(* PLC project RobotLibrary, Beckhoff Automation GmbH TwinCAT PLC Control 3.5.13.21 *)
(* stored: creationDateTime 2024-06-05T21:41:09.5070225, modificationDateTime 2024-06-05T21:41:09.5090704 *)

{attribute 'pack_mode' := '1'} 
// ------------------------------------------------------------------------- 
//  SRCI Robot Library                                                
// ------------------------------------------------------------------------- 
//                                                                           
//  Object:      ExecutionModeAllowed                                       
//  Author:      Thorsten Brach                                                
//  Date:        2024-06-01
//
//  Description:                                              
//   
//                                                                           
//  Copyright: 
//    (C) 2024 Thorsten Brach. All rights reserved                                                                         
//                                                                           
//  Disclaimer:                                                                           
//    This project is provided without any guarantee and can be used for   
//    private and commercial purposes. Any commercial use is at the user’s 
//    own risk and responsibility.
//
// -------------------------------------------------------------------------
TYPE ExecutionModeAllowed :
STRUCT
  ///
  PRIMARY_SEQ         : BOOL;
  ///
  PRIMARY_SEQ_ABORT   : BOOL;
  ///
  SECONDARY_SEQ       : BOOL;
  ///
  SECONDARY_SEQ_ABORT : BOOL;
  ///
  PAR                 : BOOL := TRUE;
  ///
  PAR_TASK            : BOOL;
  ///
  PAR_TRIGGER         : BOOL;
  ///
  PAR_TRIGGER_TASK    : BOOL;
END_STRUCT
END_TYPE

{attribute 'pack_mode' := '1'} 
// ------------------------------------------------------------------------- 
//  SRCI Robot Library                                                
// ------------------------------------------------------------------------- 
//                                                                           
//  Object:      MessageHeaderCommand                                       
//  Author:      Thorsten Brach                                                
//  Date:        2024-06-01
//
//  Description:                                              
//   
//                                                                           
//  Copyright: 
//    (C) 2024 Thorsten Brach. All rights reserved                                                                         
//                                                                           
//  Disclaimer:                                                                           
//    This project is provided without any guarantee and can be used for   
//    private and commercial purposes. Any commercial use is at the user’s 
//    own risk and responsibility.
//
// -------------------------------------------------------------------------
TYPE MessageHeaderCommand :
STRUCT
  /// Byte 00-01 :  CMD type as per specification
  CmdType      : CmdType;
  /// Byte 02  : ExecutionMode (Bit 0..3)
  ExecMode     : BYTE;  
  /// Byte 03 : CMD priority (Bit 0..3)
  Prio         : BYTE;
  /// Byte 03 : Parameter Sequence (Bit 4..7 )
  ParSeq       : BYTE;
  /// Trigger related EmitterID
  EmitterID    : ARRAY[0..3] OF SINT;
  /// Trigger related ListenerID 
  ListenerID   : SINT;
  /// Reserved
  Reserved     : BYTE;
  //// Payload length defined by type per CMD definition. Processed by Appl. Layer Task.
  Payload      : ARRAY[0..RobotLibraryParameter.TELEGRAM_PAYLOAD_MAX] OF BYTE;  
END_STRUCT
END_TYPE

{attribute 'pack_mode' := '1'} 
// ------------------------------------------------------------------------- 
//  SRCI Robot Library                                                
// ------------------------------------------------------------------------- 
//                                                                           
//  Object:      MessageHeaderResponse                                       
//  Author:      Thorsten Brach                                                
//  Date:        2024-06-01
//
//  Description:                                              
//   
//                                                                           
//  Copyright: 
//    (C) 2024 Thorsten Brach. All rights reserved                                                                         
//                                                                           
//  Disclaimer:                                                                           
//    This project is provided without any guarantee and can be used for   
//    private and commercial purposes. Any commercial use is at the user’s 
//    own risk and responsibility.
//
// -------------------------------------------------------------------------
TYPE MessageHeaderResponse :
STRUCT
  /// Byte 03 : CMD priority (Bit 0..3)
  Prio                    : BYTE;
  /// Byte 03 : Parameter Sequence (Bit 4..7 )
  ParSeq                  : BYTE;
  /// Alarm Message Severity
  AlarmMessageSeverity    : Severity;
  /// Alarm Message Code
  AlarmMessageCode        : UINT;
  /// Number of Trigger based CMD invocations
  InvocationCounter       : USINT;
  /// Number of missed Triggers
  MissedInvocationCounter : USINT;
  /// FollowID of Trigger initiator
  OriginID                : WORD;
  /// RSP Payload defined by type per CMD definition. Generated by Appl. Layer Task
  Payload                 : ARRAY[0..RobotLibraryParameter.TELEGRAM_PAYLOAD_MAX] OF BYTE;  
END_STRUCT
END_TYPE

{attribute 'qualified_only'}
// ------------------------------------------------------------------------- 
//  SRCI Robot Library                                                
// ------------------------------------------------------------------------- 
//                                                                           
//  Object:      ArmConfigElbow                                       
//  Author:      Thorsten Brach                                                
//  Date:        2024-06-01
//
//  Description:                                              
//   
//                                                                           
//  Copyright: 
//    (C) 2024 Thorsten Brach. All rights reserved                                                                         
//                                                                           
//  Disclaimer:                                                                           
//    This project is provided without any guarantee and can be used for   
//    private and commercial purposes. Any commercial use is at the user’s 
//    own risk and responsibility.
//
// -------------------------------------------------------------------------
TYPE ArmConfigElbow :
(
 /// Use config in position	
 USE_CONFIG := 0,
 /// Do not change config with this movement. (default)
 SAME := 1,
 /// Configuration in position is not used but the Robot is free to change config
 FREE := 2,
 /// Set elbow configuration in position to Down
 DOWN := 3,
 /// Set elbow configuration in position to up
 UP   := 4
);
END_TYPE

{attribute 'qualified_only'}
// ------------------------------------------------------------------------- 
//  SRCI Robot Library                                                
// ------------------------------------------------------------------------- 
//                                                                           
//  Object:      ArmConfigShoulder                                       
//  Author:      Thorsten Brach                                                
//  Date:        2024-06-01
//
//  Description:                                              
//   
//                                                                           
//  Copyright: 
//    (C) 2024 Thorsten Brach. All rights reserved                                                                         
//                                                                           
//  Disclaimer:                                                                           
//    This project is provided without any guarantee and can be used for   
//    private and commercial purposes. Any commercial use is at the user’s 
//    own risk and responsibility.
//
// -------------------------------------------------------------------------
TYPE ArmConfigShoulder :
(
 /// Use config in position	
 USE_CONFIG := 0,
 /// Do not change config with this movement. (default)
 SAME := 1,
 /// Configuration in position is not used but the Robot is free to change config
 FREE := 2,
 /// Set shoulder configuration in position to Back
 BACK := 3,
 /// Set shoulder configuration in position to Front
 FRONT := 4
);
END_TYPE

{attribute 'qualified_only'}
// ------------------------------------------------------------------------- 
//  SRCI Robot Library                                                
// ------------------------------------------------------------------------- 
//                                                                           
//  Object:      ArmConfigWrist                                       
//  Author:      Thorsten Brach                                                
//  Date:        2024-06-01
//
//  Description:                                              
//   
//                                                                           
//  Copyright: 
//    (C) 2024 Thorsten Brach. All rights reserved                                                                         
//                                                                           
//  Disclaimer:                                                                           
//    This project is provided without any guarantee and can be used for   
//    private and commercial purposes. Any commercial use is at the user’s 
//    own risk and responsibility.
//
// -------------------------------------------------------------------------
TYPE ArmConfigWrist :
(
 /// Use config in position	
 USE_CONFIG := 0,
 /// Do not change config with this movement. (default)
 SAME := 1,
 /// Configuration in position is not used but the Robot is free to change config
 FREE := 2,
 /// Set wrist configuration in position to Flip
 FLIP := 3,
 /// Set wrist configuration in position to Non-Flip
 NON_FLIP := 4
);
END_TYPE

{attribute 'qualified_only'}
// ------------------------------------------------------------------------- 
//  SRCI Robot Library                                                
// ------------------------------------------------------------------------- 
//                                                                           
//  Object:      SequenceFlag                                       
//  Author:      Thorsten Brach                                                
//  Date:        2024-06-01
//
//  Description:                                              
//   
//                                                                           
//  Copyright: 
//    (C) 2024 Thorsten Brach. All rights reserved                                                                         
//                                                                           
//  Disclaimer:                                                                           
//    This project is provided without any guarantee and can be used for   
//    private and commercial purposes. Any commercial use is at the user’s 
//    own risk and responsibility.
//
// -------------------------------------------------------------------------
TYPE SequenceFlag :
(
  /// • Refers to ProcessingModes 2 to 5 and 9
  /// • Command is not handled by any sequence
  /// • For more information on ProcessingModes refer to chapter 5.6.4.5
	NO_SEQUENCE        := 0,
  /// • Command will be handled by primary sequence
  PRIMARY_SEQUENCE   := 1,
  /// • Command will be handled by secondary sequence
  SECONDARY_SEQUENCE := 2
)USINT;
END_TYPE

{attribute 'qualified_only'}
// ------------------------------------------------------------------------- 
//  SRCI Robot Library                                                
// ------------------------------------------------------------------------- 
//                                                                           
//  Object:      LogLevel                                       
//  Author:      Thorsten Brach                                                
//  Date:        2024-06-01
//
//  Description:                                              
//   
//                                                                           
//  Copyright: 
//    (C) 2024 Thorsten Brach. All rights reserved                                                                         
//                                                                           
//  Disclaimer:                                                                           
//    This project is provided without any guarantee and can be used for   
//    private and commercial purposes. Any commercial use is at the user’s 
//    own risk and responsibility.
//
// -------------------------------------------------------------------------
TYPE LogLevel  :
(
  /// No events will be logged
  DEACTIVATE  := 0,
  /// Debugging messages, Informative messages, Warning messages, Error messages, Fatal error messages 
  DEBUG       := 4,
  /// Informative messages, Warning messages, Error messages, Fatal error messages
  INFO        := 5, 
  /// Warning messages, Error messages, Fatal error messages
  WARNING     := 20,
  /// Error messages, Fatal error messages 
  ERROR       := 28, 
  /// Fatal error messages
  FATAL_ERROR := 29 
)USINT;
END_TYPE

{attribute 'qualified_only'}
// ------------------------------------------------------------------------- 
//  SRCI Robot Library                                                
// ------------------------------------------------------------------------- 
//                                                                           
//  Object:      MessageLevel                                       
//  Author:      Thorsten Brach                                                
//  Date:        2024-06-01
//
//  Description:                                              
//   
//                                                                           
//  Copyright: 
//    (C) 2024 Thorsten Brach. All rights reserved                                                                         
//                                                                           
//  Disclaimer:                                                                           
//    This project is provided without any guarantee and can be used for   
//    private and commercial purposes. Any commercial use is at the user’s 
//    own risk and responsibility.
//
// -------------------------------------------------------------------------
TYPE MessageLevel :
(
  /// Debugging messages, Informative messages, Warning messages, Error messages, Fatal error messages
	DEBUG := 4,
  /// Informative messages, Warning messages, Error messages, Fatal error messages 
  INFO := 5, 
  /// Warning messages, Error messages, Fatal error messages
  WARNING := 20,
  /// Error messages, Fatal error messages 
  ERROR := 28 
)USINT;
END_TYPE

{attribute 'qualified_only'}
// ------------------------------------------------------------------------- 
//  SRCI Robot Library                                                
// ------------------------------------------------------------------------- 
//                                                                           
//  Object:      PriorityLevel                                       
//  Author:      Thorsten Brach                                                
//  Date:        2024-06-01
//
//  Description:                                              
//   
//                                                                           
//  Copyright: 
//    (C) 2024 Thorsten Brach. All rights reserved                                                                         
//                                                                           
//  Disclaimer:                                                                           
//    This project is provided without any guarantee and can be used for   
//    private and commercial purposes. Any commercial use is at the user’s 
//    own risk and responsibility.
//
// -------------------------------------------------------------------------
TYPE PriorityLevel :
(
  /// priority level is very high 
	VERY_HIGH := 1,
  /// priority level is high 
  HIGH      := 2,
  /// priority level is normal 
	NORMAL    := 3,
  /// priority level is low 
	LOW       := 4  
)BYTE;
END_TYPE

{attribute 'qualified_only'}
{attribute 'strict'}
// ------------------------------------------------------------------------- 
//  SRCI Robot Library                                                
// ------------------------------------------------------------------------- 
//                                                                           
//  Object:      CircPlane                                       
//  Author:      Thorsten Brach                                                
//  Date:        2024-06-01
//
//  Description:                                              
//   
//                                                                           
//  Copyright: 
//    (C) 2024 Thorsten Brach. All rights reserved                                                                         
//                                                                           
//  Disclaimer:                                                                           
//    This project is provided without any guarantee and can be used for   
//    private and commercial purposes. Any commercial use is at the user’s 
//    own risk and responsibility.
//
// -------------------------------------------------------------------------
TYPE CircPlane :
(
  /// x-z-plane
	XZ_PLANE := 0,
  /// y-z-plane
  YZ_PLANE := 1,
  /// x-y-plane
  XY_PLANE := 2
)SINT;
END_TYPE

{attribute 'qualified_only'}
// ------------------------------------------------------------------------- 
//  SRCI Robot Library                                                
// ------------------------------------------------------------------------- 
//                                                                           
//  Object:      ControlHalfByte                                       
//  Author:      Thorsten Brach                                                
//  Date:        2024-06-01
//
//  Description:                                              
//   
//                                                                           
//  Copyright: 
//    (C) 2024 Thorsten Brach. All rights reserved                                                                         
//                                                                           
//  Disclaimer:                                                                           
//    This project is provided without any guarantee and can be used for   
//    private and commercial purposes. Any commercial use is at the user’s 
//    own risk and responsibility.
//
// -------------------------------------------------------------------------
TYPE ControlHalfByte :
(
  /// Default value, no control active
  NONE := 0,
  /// Initialization is requested by the client
  INITIALIZE := 1,
  /// Resume of operation is requested by the client
  RESUME := 2,
  /// Resetting of the RC is requested by the client. The RC must stop the motion, and clear all state.
  RESET := 3,
  /// Acknowledgement of a telegram state error
  ACK_ERROR := 4,
  /// Signaling that a client error occurred. The Server must respond by setting its RI state to NOT_INITIALIZED
  CLIENT_ERROR := 5
)BYTE;
END_TYPE

{attribute 'qualified_only'}
// ------------------------------------------------------------------------- 
//  SRCI Robot Library                                                
// ------------------------------------------------------------------------- 
//                                                                           
//  Object:      ErrorReaction                                       
//  Author:      Thorsten Brach                                                
//  Date:        2024-06-01
//
//  Description:                                              
//   
//                                                                           
//  Copyright: 
//    (C) 2024 Thorsten Brach. All rights reserved                                                                         
//                                                                           
//  Disclaimer:                                                                           
//    This project is provided without any guarantee and can be used for   
//    private and commercial purposes. Any commercial use is at the user’s 
//    own risk and responsibility.
//
// -------------------------------------------------------------------------
TYPE ErrorReaction :
(
  /// Abort and move Abort active move command and delete commands buffered in sequence Move robot by specified ErrorVector
  ABORT_AND_MOVE := 0,
  /// 1: Abort
  /// Abort active move command and delete commands buffered in sequence
  /// No additional movements
  ABORT := 1,  
  /// 2: No reaction
  /// Error event is ignored by active move command
  NO_REACTION := 2
)USINT;
END_TYPE

{attribute 'qualified_only'}
// ------------------------------------------------------------------------- 
//  SRCI Robot Library                                                
// ------------------------------------------------------------------------- 
//                                                                           
//  Object:      LoadMeasurementSteps                                       
//  Author:      Thorsten Brach                                                
//  Date:        2024-06-01
//
//  Description:                                              
//   
//                                                                           
//  Copyright: 
//    (C) 2024 Thorsten Brach. All rights reserved                                                                         
//                                                                           
//  Disclaimer:                                                                           
//    This project is provided without any guarantee and can be used for   
//    private and commercial purposes. Any commercial use is at the user’s 
//    own risk and responsibility.
//
// -------------------------------------------------------------------------
TYPE LoadMeasurementSteps :
(
  /// • 0: Reset (default)
  /// Delete all positions saved on the RC
  RESET := 0,  
  /// • 1: First position
  /// Save the first position for the load estimation with the required data
  FIRST_POSITION := 1,  
  /// • 2: Second position
  /// Save the second position for the load estimation with the required data
  SECOND_POSITION := 2,  
  /// • 3: Third position
  /// Save the third position for the load estimation with the required data
  THIRD_POSITION := 3,  
  /// • 4: Fourth position
  /// Save the fourth position for the load estimation with the required data
  FOURTH_POSITION := 4,  
  /// • 99: Load calculation
  /// Start the load calculation with the data saved in the four positions
  LOAD_CALCULATION := 99
);
END_TYPE

{attribute 'qualified_only'}
// ------------------------------------------------------------------------- 
//  SRCI Robot Library                                                
// ------------------------------------------------------------------------- 
//                                                                           
//  Object:      PathChoice                                       
//  Author:      Thorsten Brach                                                
//  Date:        2024-06-01
//
//  Description:                                              
//   
//                                                                           
//  Copyright: 
//    (C) 2024 Thorsten Brach. All rights reserved                                                                         
//                                                                           
//  Disclaimer:                                                                           
//    This project is provided without any guarantee and can be used for   
//    private and commercial purposes. Any commercial use is at the user’s 
//    own risk and responsibility.
//
// -------------------------------------------------------------------------
TYPE PathChoice :
(
  /// Clockwise movement of the circular path
	CLOCKWISE := 0,
  /// Counterclockwise movement of the circular path
	COUNTERCLOCKWISE := 1
)BYTE;
END_TYPE

{attribute 'qualified_only'}
// ------------------------------------------------------------------------- 
//  SRCI Robot Library                                                
// ------------------------------------------------------------------------- 
//                                                                           
//  Object:      ReferenceElement                                       
//  Author:      Thorsten Brach                                                
//  Date:        2024-06-01
//
//  Description:                                              
//   
//                                                                           
//  Copyright: 
//    (C) 2024 Thorsten Brach. All rights reserved                                                                         
//                                                                           
//  Disclaimer:                                                                           
//    This project is provided without any guarantee and can be used for   
//    private and commercial purposes. Any commercial use is at the user’s 
//    own risk and responsibility.
//
// -------------------------------------------------------------------------
TYPE ReferenceElement :
(
  /// 0 (default): Not used
  NOT_USED := 0,  
  /// 1: X-Axis
  X_AXIS := 1,
  /// 2: Y-Axis
  Y_AXIS := 2,
  /// 3: Z-Axis
  Z_AXIS := 3,
  /// 4: XY-Plane
  XY_PLANE := 4,
  /// 5: XZ-Plane
  XZ_PLANE := 5,
  /// 6: YZ-Plane
  YZ_PLANE := 6
);
END_TYPE

{attribute 'qualified_only'}
// ------------------------------------------------------------------------- 
//  SRCI Robot Library                                                
// ------------------------------------------------------------------------- 
//                                                                           
//  Object:      Severity                                       
//  Author:      Thorsten Brach                                                
//  Date:        2024-06-01
//
//  Description:                                              
//   
//                                                                           
//  Copyright: 
//    (C) 2024 Thorsten Brach. All rights reserved                                                                         
//                                                                           
//  Disclaimer:                                                                           
//    This project is provided without any guarantee and can be used for   
//    private and commercial purposes. Any commercial use is at the user’s 
//    own risk and responsibility.
//
// -------------------------------------------------------------------------
TYPE Severity :
(
  /// Debug message
  /// • No user action required
  DEBUG := 4, 
  /// Informative message
  /// • No user action required
  INFO := 5,
  /// Warning message
  /// • User action will be required at some point
  WARNING := 20,
  /// Error message
  /// • User action required immediately
  ERROR := 28,
  ///  Fatal error message
  /// • User action required immediately
  /// • Reinitialization OF RI required
  FATAL_ERROR := 29
)USINT;
END_TYPE

{attribute 'qualified_only'}
// ------------------------------------------------------------------------- 
//  SRCI Robot Library                                                
// ------------------------------------------------------------------------- 
//                                                                           
//  Object:      SyncDirection                                       
//  Author:      Thorsten Brach                                                
//  Date:        2024-06-01
//
//  Description:                                              
//   
//                                                                           
//  Copyright: 
//    (C) 2024 Thorsten Brach. All rights reserved                                                                         
//                                                                           
//  Disclaimer:                                                                           
//    This project is provided without any guarantee and can be used for   
//    private and commercial purposes. Any commercial use is at the user’s 
//    own risk and responsibility.
//
// -------------------------------------------------------------------------
TYPE SyncDirection :
(
  /// No synchronization will be executed
  NO_SYNC := 0,
  /// Server data will be overwritten immediately by client data
  PLC_TO_ROB := 1,
  /// Client data will be overwritten immediately by server data
  ROB_TO_PLC := 2,
  /// Server or client data will be overwritten immediately by changed data
  AUTOMATIC  := 3
);
END_TYPE

{attribute 'qualified_only'}
// ------------------------------------------------------------------------- 
//  SRCI Robot Library                                                
// ------------------------------------------------------------------------- 
//                                                                           
//  Object:      SyncReaction                                       
//  Author:      Thorsten Brach                                                
//  Date:        2024-06-01
//
//  Description:                                              
//   
//                                                                           
//  Copyright: 
//    (C) 2024 Thorsten Brach. All rights reserved                                                                         
//                                                                           
//  Disclaimer:                                                                           
//    This project is provided without any guarantee and can be used for   
//    private and commercial purposes. Any commercial use is at the user’s 
//    own risk and responsibility.
//
// -------------------------------------------------------------------------
TYPE SyncReaction :
(
  /// • System behavior unaffected
	NO_REACTION := 0,
  /// • No automatic disable
  /// • Reaction will only apply when RA is disabled
  /// • RA can only be enabled if client and server are synchronized
  REACTION_TYPE_1 := 1,  
  /// • No automatic disable
  /// • RA can only be enabled if client and server are synchronized
  /// • RA sequence state will change to interrupted when no command is buffered in the active sequence
  /// • Continuation is only possible if client and server are synchronized
  REACTION_TYPE_2 := 2,  
  /// • No automatic disable
  /// • RA can only be enabled if client and server are synchronized
  /// • RA sequence state will change to interrupted
  /// • Continuation is only possible if client and server are synchronized
  REACTION_TYPE_3 := 3
)USINT;
END_TYPE

{attribute 'qualified_only'}
// ------------------------------------------------------------------------- 
//  SRCI Robot Library                                                
// ------------------------------------------------------------------------- 
//                                                                           
//  Object:      TriggerCondition                                       
//  Author:      Thorsten Brach                                                
//  Date:        2024-06-01
//
//  Description:                                              
//   
//                                                                           
//  Copyright: 
//    (C) 2024 Thorsten Brach. All rights reserved                                                                         
//                                                                           
//  Disclaimer:                                                                           
//    This project is provided without any guarantee and can be used for   
//    private and commercial purposes. Any commercial use is at the user’s 
//    own risk and responsibility.
//
// -------------------------------------------------------------------------
TYPE TriggerCondition :
(
  /// 5: Time in ms  - point reference is target position
  TARGET_POSITION_TIME_MS := -5,
  /// 4: TCP velocity in mm/s - point reference is target position
  TARGET_POSITION_TCP_VELOCITY_ABSOLUTE := -4,
  /// 3: TCP velocity in % of reference velocity - point reference is target position
  TARGET_POSITION_TCP_VELOCITY_PERCENT := -3,
  /// 2: Distance in mm of trajectory - point reference is target position
  TARGET_POSITION_DISTANCE_ABSOLUTE := -2,
  /// 1: Distance in % of trajectory - point reference is target position
  TARGET_POSITION_DISTANCE_PERCENT := -1,
  /// 0: Undfined 
  UNDEFINED := 0,
  /// 1: Distance in % of trajectory - point reference is start position
  START_POSITION_DISTANCE_PERCENT := 1,
  /// 2: Distance in mm of trajectory - point reference is start position
  START_POSITION_DISTANCE_ABSOLUTE := 2,
  /// 3: TCP velocity in % of reference velocity - point reference is start position
  START_POSITION_TCP_VELOCITY_PERCENT := 3,
  /// 4: TCP velocity in mm/s - point reference is start position
  START_POSITION_TCP_VELOCIT_ABSOLUTE := 4,
  /// 5: Time in ms - point reference is start position
  START_POSITION_TIME_MS := 5
)SINT;
END_TYPE

{attribute 'qualified_only'}
// ------------------------------------------------------------------------- 
//  SRCI Robot Library                                                
// ------------------------------------------------------------------------- 
//                                                                           
//  Object:      AbortingMode                                       
//  Author:      Thorsten Brach                                                
//  Date:        2024-06-01
//
//  Description:                                              
//   
//                                                                           
//  Copyright: 
//    (C) 2024 Thorsten Brach. All rights reserved                                                                         
//                                                                           
//  Disclaimer:                                                                           
//    This project is provided without any guarantee and can be used for   
//    private and commercial purposes. Any commercial use is at the user’s 
//    own risk and responsibility.
//
// -------------------------------------------------------------------------
TYPE AbortingMode :
(
  /// The current movement command as well as all stored movements are executed as programmed. 
  /// The new motion command is queued in the motion buffer.
	BUFFER := 0,
  /// The current movement command is aborted. All buffered motion movements are discarded. 
  /// The new target position is approached, depending on the motion command.
  ABORT  := 1
)SINT;
END_TYPE

{attribute 'qualified_only'}
// ------------------------------------------------------------------------- 
//  SRCI Robot Library                                                
// ------------------------------------------------------------------------- 
//                                                                           
//  Object:      BlendingMode                                       
//  Author:      Thorsten Brach                                                
//  Date:        2024-06-01
//
//  Description:                                              
//   
//                                                                           
//  Copyright: 
//    (C) 2024 Thorsten Brach. All rights reserved                                                                         
//                                                                           
//  Disclaimer:                                                                           
//    This project is provided without any guarantee and can be used for   
//    private and commercial purposes. Any commercial use is at the user’s 
//    own risk and responsibility.
//
// -------------------------------------------------------------------------
TYPE BlendingMode :
(
  /// Appended, buffered, no blending
  EXACT_STOP := 0,
  /// Start blending when the defined velocity is reached
  DEFINED_VELOCITY := 2,
  /// Define blending sphere with radius
  CORNER_DISTANCE := 3,
  /// Define blending with deviation
  MAX_CORNER_DEVIATION := 4,
  /// Define blending sphere with 2 radiuses
  CORNER_DISTANCE_2R := 10,
  /// Define blending with percentage of overlapping of deceleration and acceleration ramp
  RAMP_OVERLAP := 11,
  /// Define blending sphere with starting radius
  CORNER_DISTANCE_1R := 12
)SINT;
END_TYPE

{attribute 'qualified_only'}
// ------------------------------------------------------------------------- 
//  SRCI Robot Library                                                
// ------------------------------------------------------------------------- 
//                                                                           
//  Object:      CircMode                                       
//  Author:      Thorsten Brach                                                
//  Date:        2024-06-01
//
//  Description:                                              
//   
//                                                                           
//  Copyright: 
//    (C) 2024 Thorsten Brach. All rights reserved                                                                         
//                                                                           
//  Disclaimer:                                                                           
//    This project is provided without any guarantee and can be used for   
//    private and commercial purposes. Any commercial use is at the user’s 
//    own risk and responsibility.
//
// -------------------------------------------------------------------------
TYPE CircMode :
(
  /// "AuxPoint" defines a point on the circle crossed on the path from the starting to the end point.
  BORDER := 0,
  /// "AuxPoint" defines the center point of the circle.
  CENTER := 1,
  /// "AuxPoint" defines the center point of the circle, "Angle" defines the end position of the circular motion, and "CircPlane" defines the circle’s plane.
  CENTER_WITH_ANGLE := 2,
  /// "AuxPoint" defines a vector which length is the radius of the circle. The plane of the circle is defined by the rule of right thumb while the "AuxPoint" defines the spearhead point of the perpendicular.
  RADIUS := 3
)SINT;
END_TYPE

{attribute 'qualified_only'}
// ------------------------------------------------------------------------- 
//  SRCI Robot Library                                                
// ------------------------------------------------------------------------- 
//                                                                           
//  Object:      CollisionReactionMode                                       
//  Author:      Thorsten Brach                                                
//  Date:        2024-06-01
//
//  Description:                                              
//   
//                                                                           
//  Copyright: 
//    (C) 2024 Thorsten Brach. All rights reserved                                                                         
//                                                                           
//  Disclaimer:                                                                           
//    This project is provided without any guarantee and can be used for   
//    private and commercial purposes. Any commercial use is at the user’s 
//    own risk and responsibility.
//
// -------------------------------------------------------------------------
TYPE CollisionReactionMode :
(
  /// Standing still
	STANDING_STILL := 0,
  /// Reversed movement
  REVERSED_MOVEMENT := 1
);
END_TYPE

{attribute 'qualified_only'}
// ------------------------------------------------------------------------- 
//  SRCI Robot Library                                                
// ------------------------------------------------------------------------- 
//                                                                           
//  Object:      ConnectionMode                                       
//  Author:      Thorsten Brach                                                
//  Date:        2024-06-01
//
//  Description:                                              
//   
//                                                                           
//  Copyright: 
//    (C) 2024 Thorsten Brach. All rights reserved                                                                         
//                                                                           
//  Disclaimer:                                                                           
//    This project is provided without any guarantee and can be used for   
//    private and commercial purposes. Any commercial use is at the user’s 
//    own risk and responsibility.
//
// -------------------------------------------------------------------------
TYPE ConnectionMode :
(
  /// Encoder is connected to RC
	RC_CONNECTED := 0,
  /// Encoder is connected to PLC
  PLC_CONNECTED := 1
);
END_TYPE

{attribute 'qualified_only'}
// ------------------------------------------------------------------------- 
//  SRCI Robot Library                                                
// ------------------------------------------------------------------------- 
//                                                                           
//  Object:      DefinitionMode                                       
//  Author:      Thorsten Brach                                                
//  Date:        2024-06-01
//
//  Description:                                              
//   
//                                                                           
//  Copyright: 
//    (C) 2024 Thorsten Brach. All rights reserved                                                                         
//                                                                           
//  Disclaimer:                                                                           
//    This project is provided without any guarantee and can be used for   
//    private and commercial purposes. Any commercial use is at the user’s 
//    own risk and responsibility.
//
// -------------------------------------------------------------------------
TYPE DefinitionMode :
(
  /// ZeroPoint describes center point of body 
  Center := 1,
  /// ZeroPoint describes point on face of body. Parameter values for X2, Y2, Z2 will be ignored  
  Face   := 2 
)USINT;
END_TYPE

{attribute 'qualified_only'}
// ------------------------------------------------------------------------- 
//  SRCI Robot Library                                                
// ------------------------------------------------------------------------- 
//                                                                           
//  Object:      DetectionMode                                       
//  Author:      Thorsten Brach                                                
//  Date:        2024-06-01
//
//  Description:                                              
//   
//                                                                           
//  Copyright: 
//    (C) 2024 Thorsten Brach. All rights reserved                                                                         
//                                                                           
//  Disclaimer:                                                                           
//    This project is provided without any guarantee and can be used for   
//    private and commercial purposes. Any commercial use is at the user’s 
//    own risk and responsibility.
//
// -------------------------------------------------------------------------
TYPE DetectionMode :
(
  /// Torque (default)
	TORQUE := 0,
  /// Force
  FORCE := 1,
  /// Electrical current
  ELECTRICAL_CURRENT := 2,
  /// Following Error
  FOLLOWING_ERROR := 3
)USINT;
END_TYPE

{attribute 'qualified_only'}
// ------------------------------------------------------------------------- 
//  SRCI Robot Library                                                
// ------------------------------------------------------------------------- 
//                                                                           
//  Object:      ErrorTriggerMode                                       
//  Author:      Thorsten Brach                                                
//  Date:        2024-06-01
//
//  Description:                                              
//   
//                                                                           
//  Copyright: 
//    (C) 2024 Thorsten Brach. All rights reserved                                                                         
//                                                                           
//  Disclaimer:                                                                           
//    This project is provided without any guarantee and can be used for   
//    private and commercial purposes. Any commercial use is at the user’s 
//    own risk and responsibility.
//
// -------------------------------------------------------------------------
TYPE ErrorTriggerMode :
(
  /// Any command (default)
  ANY_COMMAND := 0,
  /// General commands
  GENERAL_COMMANDS := 1,
  /// Administrative commands
  ADMINISTRATIVE_COMMANDS := 2,
  /// Move commands
  MOVE_COMMANDS := 3,
  /// Periphery commands
  PERIPHERY_COMMANDS := 4,
  /// Extended commands
  EXTENDED_COMMANDS := 5,
  /// Specific command or RI message
  SPECIFIC_COMMAND_OR_RI_MESSAGE := 6,
  /// Specific RC or RA message code
  SPECIFIC_RC_OR_RA_MESSAGE_CODE := 7,
  /// Any RI message code
  ANY_RI_MESSAGE_CODE := 8,
  /// Any RC or RA message code
  ANY_RC_OR_RA_MESSAGE_CODE := 9
)SINT;
END_TYPE

{attribute 'qualified_only'}
// ------------------------------------------------------------------------- 
//  SRCI Robot Library                                                
// ------------------------------------------------------------------------- 
//                                                                           
//  Object:      ExecutionMode                                       
//  Author:      Thorsten Brach                                                
//  Date:        2024-06-01
//
//  Description:                                              
//   
//                                                                           
//  Copyright: 
//    (C) 2024 Thorsten Brach. All rights reserved                                                                         
//                                                                           
//  Disclaimer:                                                                           
//    This project is provided without any guarantee and can be used for   
//    private and commercial purposes. Any commercial use is at the user’s 
//    own risk and responsibility.
//
// -------------------------------------------------------------------------
TYPE ExecutionMode :
(
  /// Command is buffered in sequence buffer and executed once
  SEQUENCE_PRIMARY := 0,
  /// Command is buffered in sequence buffer, aborts and empties previous commands in sequence buffer, and is executed once
  SEQUENCE_ABORT_OTHERS_PRIMARY := 1,
  /// Command is buffered in parallel buffer and executed once. The execution may also be Trigger based.
  PARALLEL := 2,
  /// Command is buffered in parallel buffer and executed repeatedly until deliberate deactivation by user. The de- and activation may also be Trigger based.
  CONTINUOUS := 3,
  /// Command is buffered and executed once when triggered. The CMD remains in the buffer until removed by the user.
  TRIGGER_MULTIPLE := 5,
  /// Command is buffered in sequence buffer and executed once (Secondary)
  SEQUENCE_SECONDARY := 7,
  /// Command is buffered in sequence buffer, aborts and empties previous commands in sequence buffer and is executed once (Secondary)
  SEQUENCE_ABORT_OTHERS_SECONDARY := 8,
  /// CMD execution is stopped and/or CMD is removed from the buffer.
  STOP_PARALLEL_CONTINUOUS_TRIGGER := 9
)USINT;
END_TYPE

{attribute 'qualified_only'}
// ------------------------------------------------------------------------- 
//  SRCI Robot Library                                                
// ------------------------------------------------------------------------- 
//                                                                           
//  Object:      FrameCalculationMode                                       
//  Author:      Thorsten Brach                                                
//  Date:        2024-06-01
//
//  Description:                                              
//   
//                                                                           
//  Copyright: 
//    (C) 2024 Thorsten Brach. All rights reserved                                                                         
//                                                                           
//  Disclaimer:                                                                           
//    This project is provided without any guarantee and can be used for   
//    private and commercial purposes. Any commercial use is at the user’s 
//    own risk and responsibility.
//
// -------------------------------------------------------------------------
TYPE FrameCalculationMode :
(
  /// 0: Three-Point-method (default)
  THREE_POINT_METHOD := 0,  
  /// 1: Four-Point-method
  FOUR_POINT_METHOD := 1,  
  /// 2: One-Point-method
  ONE_POINT_METHOD := 2
)SINT;
END_TYPE

{attribute 'qualified_only'}
// ------------------------------------------------------------------------- 
//  SRCI Robot Library                                                
// ------------------------------------------------------------------------- 
//                                                                           
//  Object:      FunctionMode                                       
//  Author:      Thorsten Brach                                                
//  Date:        2024-06-01
//
//  Description:                                              
//   
//                                                                           
//  Copyright: 
//    (C) 2024 Thorsten Brach. All rights reserved                                                                         
//                                                                           
//  Disclaimer:                                                                           
//    This project is provided without any guarantee and can be used for   
//    private and commercial purposes. Any commercial use is at the user’s 
//    own risk and responsibility.
//
// -------------------------------------------------------------------------
TYPE FunctionMode :
(
	enum_member := 0
);
END_TYPE

{attribute 'qualified_only'}
// ------------------------------------------------------------------------- 
//  SRCI Robot Library                                                
// ------------------------------------------------------------------------- 
//                                                                           
//  Object:      InterpolationMode                                       
//  Author:      Thorsten Brach                                                
//  Date:        2024-06-01
//
//  Description:                                              
//   
//                                                                           
//  Copyright: 
//    (C) 2024 Thorsten Brach. All rights reserved                                                                         
//                                                                           
//  Disclaimer:                                                                           
//    This project is provided without any guarantee and can be used for   
//    private and commercial purposes. Any commercial use is at the user’s 
//    own risk and responsibility.
//
// -------------------------------------------------------------------------
TYPE InterpolationMode :
(
  /// Linear interpolation
	Linear_interpolation := 0,
  /// Direct interpolation (PTP)
  Direct_interpolation := 1
);
END_TYPE

{attribute 'qualified_only'}
// ------------------------------------------------------------------------- 
//  SRCI Robot Library                                                
// ------------------------------------------------------------------------- 
//                                                                           
//  Object:      JogMode                                       
//  Author:      Thorsten Brach                                                
//  Date:        2024-06-01
//
//  Description:                                              
//   
//                                                                           
//  Copyright: 
//    (C) 2024 Thorsten Brach. All rights reserved                                                                         
//                                                                           
//  Disclaimer:                                                                           
//    This project is provided without any guarantee and can be used for   
//    private and commercial purposes. Any commercial use is at the user’s 
//    own risk and responsibility.
//
// -------------------------------------------------------------------------
TYPE JogMode :
(
  /// • Jog TCP manually in the given frame (WCS/UCS)
  /// • Movement on several coordinate axes simultaneously possible
	JOG_FRAME := 0,
  /// • Jog TCP manually in the given tool coordinate system
  /// • Movement on several coordinate axes simultaneously possible
  JOG_TOOL := 1,
  /// • Jog joints manually without referring to a given frame or tool
  /// • Movement of several axes simultaneously possible.
  JOG_AXES := 2
)USINT;
END_TYPE

{attribute 'qualified_only'}
// ------------------------------------------------------------------------- 
//  SRCI Robot Library                                                
// ------------------------------------------------------------------------- 
//                                                                           
//  Object:      LimitMode                                       
//  Author:      Thorsten Brach                                                
//  Date:        2024-06-01
//
//  Description:                                              
//   
//                                                                           
//  Copyright: 
//    (C) 2024 Thorsten Brach. All rights reserved                                                                         
//                                                                           
//  Disclaimer:                                                                           
//    This project is provided without any guarantee and can be used for   
//    private and commercial purposes. Any commercial use is at the user’s 
//    own risk and responsibility.
//
// -------------------------------------------------------------------------
TYPE LimitMode :
(
  /// 0: No limit defined (default)
  /// The robot can be moved in the direction set with the input parameter "CompliantAxes" in a compliant manner by applying an external force on it.
  /// By reaching the mechanical or software limits, the robot stops.
  NO_LIMIT_DEFINED := 0,
  
  /// 1: Limit defined
  /// The robot can be moved along the defined vector in a compliant manner by applying an external force on it.
  /// By reaching the vector limit defined by the input parameter "VectorData", the robot stops.
  LIMIT_DEFINED := 1
)USINT;
END_TYPE

{attribute 'qualified_only'}
// ------------------------------------------------------------------------- 
//  SRCI Robot Library                                                
// ------------------------------------------------------------------------- 
//                                                                           
//  Object:      LoadMeasurementMode                                       
//  Author:      Thorsten Brach                                                
//  Date:        2024-06-01
//
//  Description:                                              
//   
//                                                                           
//  Copyright: 
//    (C) 2024 Thorsten Brach. All rights reserved                                                                         
//                                                                           
//  Disclaimer:                                                                           
//    This project is provided without any guarantee and can be used for   
//    private and commercial purposes. Any commercial use is at the user’s 
//    own risk and responsibility.
//
// -------------------------------------------------------------------------
TYPE  LoadMeasurementMode :
(
  /// 0: One Position (default)
  /// Use one defined position and optional axes ranges
  ONE_POSITION := 0,  
  /// 1: Configuration Angle
  /// Use one defined position and optional axes ranges
  CONFIGURATION_ANGLE := 1,  
  /// 2: Area
  /// Use a defined area for the measurement
  AREA := 2,  
  /// 3: Two Positions
  /// Use defined positions for the measurement
  TWO_POSITIONS := 3
)USINT;
END_TYPE

{attribute 'qualified_only'}
// ------------------------------------------------------------------------- 
//  SRCI Robot Library                                                
// ------------------------------------------------------------------------- 
//                                                                           
//  Object:      LogonMode                                       
//  Author:      Thorsten Brach                                                
//  Date:        2024-06-01
//
//  Description:                                              
//   
//                                                                           
//  Copyright: 
//    (C) 2024 Thorsten Brach. All rights reserved                                                                         
//                                                                           
//  Disclaimer:                                                                           
//    This project is provided without any guarantee and can be used for   
//    private and commercial purposes. Any commercial use is at the user’s 
//    own risk and responsibility.
//
// -------------------------------------------------------------------------
TYPE LogonMode :
(
  /// Password only (default)
	PASSWORD_ONLY := 0,
  /// Username and Password
  USERNAME_AND_PASSWORD := 1,
  /// Level ID and Password
  LEVEL_ID_AND_PASSWORD := 2
)SINT;
END_TYPE

{attribute 'qualified_only'}
// ------------------------------------------------------------------------- 
//  SRCI Robot Library                                                
// ------------------------------------------------------------------------- 
//                                                                           
//  Object:      MeasuringIoMode                                       
//  Author:      Thorsten Brach                                                
//  Date:        2024-06-01
//
//  Description:                                              
//   
//                                                                           
//  Copyright: 
//    (C) 2024 Thorsten Brach. All rights reserved                                                                         
//                                                                           
//  Disclaimer:                                                                           
//    This project is provided without any guarantee and can be used for   
//    private and commercial purposes. Any commercial use is at the user’s 
//    own risk and responsibility.
//
// -------------------------------------------------------------------------
TYPE MeasuringIoMode :
(
  /// Measurement at next rising edge 
  /// • Output "MeasuredPosition_1" used
	MEASUREMENT_AT_NEXT_RISING_EDGE := 0,
  /// Measurement at next falling edge 
  /// • Output "MeasuredPosition_1" used
  MEASUREMENT_AT_NEXT_FALLING_EDGE := 1,
  /// Measurement at next edges, regardless of rising or falling edges.
  /// • First position stored in output "MeasuredPosition_1"
  /// • Second position stored in output "MeasuredPosition_2"
  MEASUREMENT_AT_NEXT_EDGE := 2,
  /// Measurement at two edges, beginning with the rising edge:
  /// • Rising edge = "MeasuredPosition_1 "
  /// • Falling edge = "MeasuredPosition_2 "
  MEASUREMENT_AT_TWO_EDGES_BEGIN_WITH_RISING := 3,
  /// Measurement at two edges, beginning with the falling edge:
  /// • Falling edge = " MeasuredPosition_1 "
  /// • Rising edge = "MeasuredPosition_2 "
  MEASUREMENT_AT_TWO_EDGES_BEGIN_WITH_FALLING := 4
);
END_TYPE

{attribute 'qualified_only'}
// ------------------------------------------------------------------------- 
//  SRCI Robot Library                                                
// ------------------------------------------------------------------------- 
//                                                                           
//  Object:      MeasuringUnitMode                                       
//  Author:      Thorsten Brach                                                
//  Date:        2024-06-01
//
//  Description:                                              
//   
//                                                                           
//  Copyright: 
//    (C) 2024 Thorsten Brach. All rights reserved                                                                         
//                                                                           
//  Disclaimer:                                                                           
//    This project is provided without any guarantee and can be used for   
//    private and commercial purposes. Any commercial use is at the user’s 
//    own risk and responsibility.
//
// -------------------------------------------------------------------------
TYPE MeasuringUnitMode :
(
	/// 0: VectorLength (default)
  ///    Defines the distance in millimeter between two points in cartesian space.
  VECTOR_LENGTH  := 0,
  /// 1: SegmentLength
  ///    Defines the distance in mm covered between the two points in cartesian space
  SEGMENT_LENGTH := 1,
  /// 2: Time
  ///    Defines the duration in milliseconds between the start and end point.
  TIME_DURATION  := 2
)USINT;
END_TYPE

{attribute 'qualified_only'}
// ------------------------------------------------------------------------- 
//  SRCI Robot Library                                                
// ------------------------------------------------------------------------- 
//                                                                           
//  Object:      OperationMode                                       
//  Author:      Thorsten Brach                                                
//  Date:        2024-06-01
//
//  Description:                                              
//   
//                                                                           
//  Copyright: 
//    (C) 2024 Thorsten Brach. All rights reserved                                                                         
//                                                                           
//  Disclaimer:                                                                           
//    This project is provided without any guarantee and can be used for   
//    private and commercial purposes. Any commercial use is at the user’s 
//    own risk and responsibility.
//
// -------------------------------------------------------------------------
TYPE OperationMode :
(
 /// Test mode 1:
 /// • Maximum velocity of TCP is restricted to <250 mm/s
 /// • Robot can only be moved while enable switch is active
 /// • Designed for jogging, teaching program, verification
 /// • Safety door can be opened
 T1_LOCAL := 1,
 /// Test mode 2:
 /// • Maximum velocity of TCP not restricted (100%)
 /// • Robot can only be moved while enable switch is active
 /// • Designed for program verification (step mode)
 /// • Safety door can be opened
 T2_LOCAL := 2,
 /// Automatic mode:
 /// • Maximum velocity of TCP not restricted (100%)
 /// • Robot is executing user program automatically
 /// • Robot will stop if safety devices report error (e.g. safety door must be closed)
 AUTO := 3,
 /// External Automatic mode (PLC mode)
 /// • Robot is operated remotely only
 /// • Maximum velocity of TCP not restricted (100%)
 /// • Robot is executing user program automatically
 /// • Jogging possible
 /// • Robot will stop if safety devices report error (e.g. safety door must be closed)
 AUTO_EXT := 4,
 /// External Test mode 1 (PLC mode with T1 functionality)
 /// • Robot is operated remotely only
 /// • Maximum velocity of TCP is restricted to <250 mm/s
 /// • Robot can only be moved while enable switch is active
 /// • Designed for jogging, teaching, program verification
 /// • Safety door can be opened
 T1_EXT := 5,
 /// External Test mode 2:
 /// • Robot is operated remotely only
 /// • Maximum velocity of TCP not restricted (100%)
 /// • Robot can only be moved while enable switch is active
 /// • Designed for jogging, program verification (step mode)
 /// • Safety door can be opened
 T2_EXT := 6
)USINT;
END_TYPE

{attribute 'qualified_only'}
// ------------------------------------------------------------------------- 
//  SRCI Robot Library                                                
// ------------------------------------------------------------------------- 
//                                                                           
//  Object:      OrientationMode                                       
//  Author:      Thorsten Brach                                                
//  Date:        2024-06-01
//
//  Description:                                              
//   
//                                                                           
//  Copyright: 
//    (C) 2024 Thorsten Brach. All rights reserved                                                                         
//                                                                           
//  Disclaimer:                                                                           
//    This project is provided without any guarantee and can be used for   
//    private and commercial purposes. Any commercial use is at the user’s 
//    own risk and responsibility.
//
// -------------------------------------------------------------------------
TYPE OrientationMode :
(
    /// Change orientation continuously in a linear way
    LINEAR_INTERPOLATED := 1,
    /// Change orientation continuously in a joint interpolated way of wrist joints
    JOINT_INTERPOLATED := 2,
    /// No change of orientation during movement
    FIX := 3,
    /// No change of orientation in relation to trajectory
    PATH := 4
)SINT;
END_TYPE

{attribute 'qualified_only'}
// ------------------------------------------------------------------------- 
//  SRCI Robot Library                                                
// ------------------------------------------------------------------------- 
//                                                                           
//  Object:      OriMode                                       
//  Author:      Thorsten Brach                                                
//  Date:        2024-06-01
//
//  Description:                                              
//   
//                                                                           
//  Copyright: 
//    (C) 2024 Thorsten Brach. All rights reserved                                                                         
//                                                                           
//  Disclaimer:                                                                           
//    This project is provided without any guarantee and can be used for   
//    private and commercial purposes. Any commercial use is at the user’s 
//    own risk and responsibility.
//
// -------------------------------------------------------------------------
TYPE OriMode :
(
  /// Change orientation continuously in a linear way
	LINEAR_INTERPOLATED := 1,
  /// Change orientation continuously in a joint interpolated way.
  JOINT_INTERPOLATED  := 2,
  /// No change of orientation during movement
  FIX                 := 3,
  /// No change of orientation in relation to trajectory
  PATH                := 4
)USINT;
END_TYPE

{attribute 'qualified_only'}
// ------------------------------------------------------------------------- 
//  SRCI Robot Library                                                
// ------------------------------------------------------------------------- 
//                                                                           
//  Object:      ProcessingMode                                       
//  Author:      Thorsten Brach                                                
//  Date:        2024-06-01
//
//  Description:                                              
//   
//                                                                           
//  Copyright: 
//    (C) 2024 Thorsten Brach. All rights reserved                                                                         
//                                                                           
//  Disclaimer:                                                                           
//    This project is provided without any guarantee and can be used for   
//    private and commercial purposes. Any commercial use is at the user’s 
//    own risk and responsibility.
//
// -------------------------------------------------------------------------
TYPE ProcessingMode :
(
  /// Command is buffered in sequence buffer and executed once
  BUFFERED := 0,
  /// Command is buffered in sequence buffer, aborts and empties previous commands in sequence buffer, and is executed once
  ABORTING := 1,
  /// Command is buffered in parallel buffer and executed once
  PARALLEL := 2,
  /// Command is buffered in parallel buffer and executed repeatedly until deliberate deactivation by user
  CONTINUOUS := 3,
  /// CMD execution is stopped and/or CMD is removed from the buffer
  DEACTIVATE := 9,
  /// Command is buffered in sequence buffer and executed once (Trigger based)
  TRIGGER_BUFFERED := 10,
  /// Command is buffered in sequence buffer, aborts and empties previous commands in sequence buffer, and is executed once (Trigger based)
  TRIGGER_ABORTING := 11,
  /// Command is buffered in parallel buffer and executed once (Trigger based)
  TRIGGER_ONCE := 12,
  /// Command is buffered in parallel buffer and executed repeatedly until deliberate deactivation by user (Trigger based)
  TRIGGER_CONTINUOUS := 13,
  /// Command is buffered and executed multiple times when triggered. The CMD remains in the buffer until removed by the user.
  TRIGGER_MULTIPLE := 14
)USINT;
END_TYPE

{attribute 'qualified_only'}
// ------------------------------------------------------------------------- 
//  SRCI Robot Library                                                
// ------------------------------------------------------------------------- 
//                                                                           
//  Object:      ResistanceForceMode                                       
//  Author:      Thorsten Brach                                                
//  Date:        2024-06-01
//
//  Description:                                              
//   
//                                                                           
//  Copyright: 
//    (C) 2024 Thorsten Brach. All rights reserved                                                                         
//                                                                           
//  Disclaimer:                                                                           
//    This project is provided without any guarantee and can be used for   
//    private and commercial purposes. Any commercial use is at the user’s 
//    own risk and responsibility.
//
// -------------------------------------------------------------------------
TYPE ResistanceForceMode :
(
  /// 0 (default): ResistanceForceTCP.
  /// Set "0" to set the resistance of the RA against the external force at the TCP.
  RESISTANCE_FORCE_TCP := 0,
  
  /// 1: ResistanceForceAxis.
  /// Set "1" to set the resistance of the RA against the external force for each axis independently.
  RESISTANCE_FORCE_AXIS := 1
)USINT;
END_TYPE

{attribute 'qualified_only'}
// ------------------------------------------------------------------------- 
//  SRCI Robot Library                                                
// ------------------------------------------------------------------------- 
//                                                                           
//  Object:      SensorConnectionMode                                       
//  Author:      Thorsten Brach                                                
//  Date:        2024-06-01
//
//  Description:                                              
//   
//                                                                           
//  Copyright: 
//    (C) 2024 Thorsten Brach. All rights reserved                                                                         
//                                                                           
//  Disclaimer:                                                                           
//    This project is provided without any guarantee and can be used for   
//    private and commercial purposes. Any commercial use is at the user’s 
//    own risk and responsibility.
//
// -------------------------------------------------------------------------
TYPE SensorConnectionMode :
(
  /// RC sensor and algorithm
  /// Force-Torque-Sensor connected to RC
  /// Control algorithm in RC
  RC_SENSOR_ALGORITHM := 0,
  
  /// PLC sensor and RC algorithm
  /// Force-Torque-Sensor connected to PLC
  /// Control algorithm in RC
  PLC_SENSOR_RC_ALGORITHM := 1,
  
  /// PLC sensor and algorithm
  /// Force-Torque-Sensor connected to PLC
  /// Control algorithm in PLC
  PLC_SENSOR_ALGORITHM := 2
)USINT;
END_TYPE

{attribute 'qualified_only'}
// ------------------------------------------------------------------------- 
//  SRCI Robot Library                                                
// ------------------------------------------------------------------------- 
//                                                                           
//  Object:      SingularityAvoidanceMode                                       
//  Author:      Thorsten Brach                                                
//  Date:        2024-06-01
//
//  Description:                                              
//   
//                                                                           
//  Copyright: 
//    (C) 2024 Thorsten Brach. All rights reserved                                                                         
//                                                                           
//  Disclaimer:                                                                           
//    This project is provided without any guarantee and can be used for   
//    private and commercial purposes. Any commercial use is at the user’s 
//    own risk and responsibility.
//
// -------------------------------------------------------------------------
TYPE SingularityAvoidanceMode :
(
  /// 0: NoChange (default)
  /// Allow movement of one or more joints to avoid singularities without a change of the orientation
  NO_CHANGE := 0,
  
  /// 1: Lock J4
  /// Lock the 4th joint to avoid singularities
  LOCK_J4 := 1,
  
  /// 2: ToolOrientation
  /// Allow a small movement of the tool orientation to avoid singularities
  TOOL_ORIENTATION := 2
)USINT;
END_TYPE

{attribute 'qualified_only'}
// ------------------------------------------------------------------------- 
//  SRCI Robot Library                                                
// ------------------------------------------------------------------------- 
//                                                                           
//  Object:      SplineMode                                       
//  Author:      Thorsten Brach                                                
//  Date:        2024-06-01
//
//  Description:                                              
//   
//                                                                           
//  Copyright: 
//    (C) 2024 Thorsten Brach. All rights reserved                                                                         
//                                                                           
//  Disclaimer:                                                                           
//    This project is provided without any guarantee and can be used for   
//    private and commercial purposes. Any commercial use is at the user’s 
//    own risk and responsibility.
//
// -------------------------------------------------------------------------
TYPE SplineMode :
(
  /// 0: Discrete Points
  DISCRETE_POINTS := 0,
  /// 1: Bézier Spline
  BEZIER_SPLINE := 1,
  /// 2: B-Splines
  B_SPLINES := 2,
  /// 3: Cubic Hermite Spline
  CUBIC_HERMITE_SPLINE := 3,
  /// 4: C-Splines
  C_SPLINES := 4
)UINT;
END_TYPE

{attribute 'qualified_only'}
// ------------------------------------------------------------------------- 
//  SRCI Robot Library                                                
// ------------------------------------------------------------------------- 
//                                                                           
//  Object:      StepMode                                       
//  Author:      Thorsten Brach                                                
//  Date:        2024-06-01
//
//  Description:                                              
//   
//                                                                           
//  Copyright: 
//    (C) 2024 Thorsten Brach. All rights reserved                                                                         
//                                                                           
//  Disclaimer:                                                                           
//    This project is provided without any guarantee and can be used for   
//    private and commercial purposes. Any commercial use is at the user’s 
//    own risk and responsibility.
//
// -------------------------------------------------------------------------
TYPE StepMode :
(
  /// StepMode is deactivated
	DEACTIVATE := 0,
  /// Blending
  /// • The robot moves on the blended trajectory
  /// • The movement is interrupted when the active segment changes
  BLENDING := 1,
  ///Exact stop
  /// • The robot moves to the defined target positions without blending
  /// • The movement is interrupted when the defined target position is reached
  EXACT_STOP := 2
)USINT;
END_TYPE

{attribute 'qualified_only'}
// ------------------------------------------------------------------------- 
//  SRCI Robot Library                                                
// ------------------------------------------------------------------------- 
//                                                                           
//  Object:      StopMode                                       
//  Author:      Thorsten Brach                                                
//  Date:        2024-06-01
//
//  Description:                                              
//   
//                                                                           
//  Copyright: 
//    (C) 2024 Thorsten Brach. All rights reserved                                                                         
//                                                                           
//  Disclaimer:                                                                           
//    This project is provided without any guarantee and can be used for   
//    private and commercial purposes. Any commercial use is at the user’s 
//    own risk and responsibility.
//
// -------------------------------------------------------------------------
TYPE StopMode :
(
  /// 0: Stop via JobID (default)
  /// TargetID is interpreted as JobID
  /// All instances of the defined JobID are stopped
  STOP_JOB_ID := 0,  
  /// 1: Stop via InstanceID
  /// TargetID is interpreted as InstanceID
  /// The instance of the defined InstanceID is stopped
  STOP_INSTANCE_ID := 1,  
  /// 2: Stop all subprograms
  /// All subprograms independent of the input parameter value of TargetID are stopped
  STOP_ALL_SUBPROGRAMS := 2
)USINT;
END_TYPE

{attribute 'qualified_only'}
// ------------------------------------------------------------------------- 
//  SRCI Robot Library                                                
// ------------------------------------------------------------------------- 
//                                                                           
//  Object:      SyncInMode                                       
//  Author:      Thorsten Brach                                                
//  Date:        2024-06-01
//
//  Description:                                              
//   
//                                                                           
//  Copyright: 
//    (C) 2024 Thorsten Brach. All rights reserved                                                                         
//                                                                           
//  Disclaimer:                                                                           
//    This project is provided without any guarantee and can be used for   
//    private and commercial purposes. Any commercial use is at the user’s 
//    own risk and responsibility.
//
// -------------------------------------------------------------------------
TYPE SyncInMode :
(
  /// • When work piece enters "SyncInZone"
  /// • Start synchronization as soon as possible within defined acceleration and velocity limits
	IN_SYNC_IN_ZONE := 0,
  /// • Start synchronization after specific distance after execution
  /// • "SynInZone" ignored
  AFTER_DISTANCE := 1,
  /// • Start synchronization after specific time after execution
  /// • "SynInZone" ignored
  AFTER_TIME := 2,
  /// • As soon as possible within defined acceleration and velocity limits
  /// • "SynInZone" ignored
  IMMEDIATELY := 3
)SINT;
END_TYPE

{attribute 'qualified_only'}
// ------------------------------------------------------------------------- 
//  SRCI Robot Library                                                
// ------------------------------------------------------------------------- 
//                                                                           
//  Object:      SyncMode                                       
//  Author:      Thorsten Brach                                                
//  Date:        2024-06-01
//
//  Description:                                              
//   
//                                                                           
//  Copyright: 
//    (C) 2024 Thorsten Brach. All rights reserved                                                                         
//                                                                           
//  Disclaimer:                                                                           
//    This project is provided without any guarantee and can be used for   
//    private and commercial purposes. Any commercial use is at the user’s 
//    own risk and responsibility.
//
// -------------------------------------------------------------------------
TYPE SyncMode :
(
  /// No synchronization will be executed
	NO_SYNCHRONIZATION := 0,
  /// Server data will be overwritten immediately by client data
  CLIENT_TO_SERVER := 1,
  /// Client data will be overwritten immediately by server data
  SERVER_TO_CLIENT := 2,
  /// Server or client data will be overwritten immediately by changed data
  AUTOMATIC := 3
)USINT;
END_TYPE

{attribute 'qualified_only'}
// ------------------------------------------------------------------------- 
//  SRCI Robot Library                                                
// ------------------------------------------------------------------------- 
//                                                                           
//  Object:      ThresholdMode                                       
//  Author:      Thorsten Brach                                                
//  Date:        2024-06-01
//
//  Description:                                              
//   
//                                                                           
//  Copyright: 
//    (C) 2024 Thorsten Brach. All rights reserved                                                                         
//                                                                           
//  Disclaimer:                                                                           
//    This project is provided without any guarantee and can be used for   
//    private and commercial purposes. Any commercial use is at the user’s 
//    own risk and responsibility.
//
// -------------------------------------------------------------------------
TYPE ThresholdMode :
(
  /// Automatic.
	Automatic := 0,
  /// Manual (according to LimitAxis)
  Manual    := 1
)USINT;
END_TYPE

{attribute 'qualified_only'}
// ------------------------------------------------------------------------- 
//  SRCI Robot Library                                                
// ------------------------------------------------------------------------- 
//                                                                           
//  Object:      ToolCalculationMode                                       
//  Author:      Thorsten Brach                                                
//  Date:        2024-06-01
//
//  Description:                                              
//   
//                                                                           
//  Copyright: 
//    (C) 2024 Thorsten Brach. All rights reserved                                                                         
//                                                                           
//  Disclaimer:                                                                           
//    This project is provided without any guarantee and can be used for   
//    private and commercial purposes. Any commercial use is at the user’s 
//    own risk and responsibility.
//
// -------------------------------------------------------------------------
TYPE ToolCalculationMode :
(
  /// 0: Two Point + Z-Method (default)
  TWO_POINT_Z_METHOD := 0,        
  /// 1: Three-Point-Method
  THREE_POINT_METHOD := 1,        
  /// 2: Four-Point-Method
  FOUR_POINT_METHOD := 2,        
  /// 3: Five-Point-Method
  FIVE_POINT_METHOD := 3,        
  /// 4: Six-Point-Method
  SIX_POINT_METHOD := 4,        
  /// 5: ABC-World-Method
  ABC_WORLD_METHOD := 5,        
  /// 6: ABC-Two-Point-Method
  ABC_TWO_POINT_METHOD := 6
)SINT;
END_TYPE

{attribute 'qualified_only'}
// ------------------------------------------------------------------------- 
//  SRCI Robot Library                                                
// ------------------------------------------------------------------------- 
//                                                                           
//  Object:      TrajectoryMode                                       
//  Author:      Thorsten Brach                                                
//  Date:        2024-06-01
//
//  Description:                                              
//   
//                                                                           
//  Copyright: 
//    (C) 2024 Thorsten Brach. All rights reserved                                                                         
//                                                                           
//  Disclaimer:                                                                           
//    This project is provided without any guarantee and can be used for   
//    private and commercial purposes. Any commercial use is at the user’s 
//    own risk and responsibility.
//
// -------------------------------------------------------------------------
TYPE TrajectoryMode :
(
  /// Invalid (default)
	INVALID := 0,
  /// Linear movement
  LINEAR_MOVEMENT := 1,
  /// PTP movement
  PTP_MOVEMENT := 2
);
END_TYPE

{attribute 'qualified_only'}
// ------------------------------------------------------------------------- 
//  SRCI Robot Library                                                
// ------------------------------------------------------------------------- 
//                                                                           
//  Object:      TransformMode                                       
//  Author:      Thorsten Brach                                                
//  Date:        2024-06-01
//
//  Description:                                              
//   
//                                                                           
//  Copyright: 
//    (C) 2024 Thorsten Brach. All rights reserved                                                                         
//                                                                           
//  Disclaimer:                                                                           
//    This project is provided without any guarantee and can be used for   
//    private and commercial purposes. Any commercial use is at the user’s 
//    own risk and responsibility.
//
// -------------------------------------------------------------------------
TYPE TransformMode :
(
  /// 0 (default): Mirror at Point with mirroring of the target position’s orientation
  /// Requires for the mirror Point the "TransformationParameter_1" and the "TransformationParameter_2" set to "Not used"
  MIRROR_AT_POINT := 0,  
  /// 1: Mirror at Straight Line with mirroring of the target position’s orientation
  /// Requires for the Straight Line the "TransformationParameter_1" and the "TransformationParameter_2" set to "X-Axis", "Y-Axis" or "Z-Axis"
  MIRROR_AT_STRAIGHT_LINE := 1,  
  /// 2: Mirror at Plane with mirroring of the target position’s orientation
  /// Requires for the Plane the "TransformationParameter_1" and the "TransformationParameter_2" set to "XY-Axis", "XZ-Axis" or "YZ-Axis"
  MIRROR_AT_PLANE := 2,  
  /// 3: Rotate around Straight Line with rotation of the target position’s orientation
  /// Requires for the Straight Line the "TransformationParameter_1" and the "TransformationParameter_2" set to "X-Axis", "Y-Axis" or "Z-Axis"
  /// Requires for the parameter "RotationAngle"
  ROTATE_AROUND_STRAIGHT_LINE := 3,  
  /// 4: Shift by Vector
  /// Requires for the shifting Vector defined by the Point the "TransformationParameter_1" and the "TransformationParameter_2" set to "Not used"
  /// Requires for the shifting shortest Vector to the Straight Line the "TransformationParameter_1" and the "TransformationParameter_2" set to "X-Axis", "Y-Axis" or "Z-Axis"
  /// Requires for the shifting shortest Vector to the Plane the "TransformationParameter_1" and the "TransformationParameter_2" set to "XY-Axis", "XZ-Axis" or "YZ-Axis"
  SHIFT_BY_VECTOR := 4
)SINT;
END_TYPE

{attribute 'qualified_only'}
// ------------------------------------------------------------------------- 
//  SRCI Robot Library                                                
// ------------------------------------------------------------------------- 
//                                                                           
//  Object:      TriggerModeIo                                       
//  Author:      Thorsten Brach                                                
//  Date:        2024-06-01
//
//  Description:                                              
//   
//                                                                           
//  Copyright: 
//    (C) 2024 Thorsten Brach. All rights reserved                                                                         
//                                                                           
//  Disclaimer:                                                                           
//    This project is provided without any guarantee and can be used for   
//    private and commercial purposes. Any commercial use is at the user’s 
//    own risk and responsibility.
//
// -------------------------------------------------------------------------
TYPE TriggerModeIo :
(
  /// Invalid (default)
  INVALID := 0,  
  /// Digital Input Rising Edge
  DIGITAL_INPUT_RISING_EDGE := 10,
  /// Digital Input Falling Edge
  DIGITAL_INPUT_FALLING_EDGE := 11,
  /// Digital Input Rising or Falling Edge
  DIGITAL_INPUT_RISING_OR_FALLING_EDGE := 12,
  /// Digital Input Rising or Falling Edge (Inverted)
  DIGITAL_INPUT_RISING_OR_FALLING_EDGE_INVERTED := 13,
  /// Digital Output Rising Edge
  DIGITAL_OUTPUT_RISING_EDGE := 20,
  /// Digital Output Falling Edge
  DIGITAL_OUTPUT_FALLING_EDGE := 21,
  /// Digital Output Rising or Falling Edge
  DIGITAL_OUTPUT_RISING_OR_FALLING_EDGE := 22,
  /// Digital Output Rising or Falling Edge (Inverted)
  DIGITAL_OUTPUT_RISING_OR_FALLING_EDGE_INVERTED := 23,
  /// Analog Input Exceeding Defined Threshold
  ANALOG_INPUT_EXCEEDING_DEFINED_THRESHOLD := 30,
  /// Analog Input Falling Below Defined Threshold
  ANALOG_INPUT_FALLING_BELOW_DEFINED_THRESHOLD := 31,
  /// Analog Input Exceeding or Falling Below Defined Threshold
  ANALOG_INPUT_EXCEEDING_OR_FALLING_BELOW_DEFINED_THRESHOLD := 32,
  /// Analog Input Exceeding or Falling Below Defined Threshold (Inverted)
  ANALOG_INPUT_EXCEEDING_OR_FALLING_BELOW_DEFINED_THRESHOLD_INVERTED := 33,
  /// Analog Input Entering Defined Range
  ANALOG_INPUT_ENTERING_DEFINED_RANGE := 34,
  /// Analog Input Leaving Defined Range
  ANALOG_INPUT_LEAVING_DEFINED_RANGE := 35,
  /// Analog Input Entering or Leaving Defined Range
  ANALOG_INPUT_ENTERING_OR_LEAVING_DEFINED_RANGE := 36,
  /// Analog Input Entering or Leaving Defined Range (Inverted)
  ANALOG_INPUT_ENTERING_OR_LEAVING_DEFINED_RANGE_INVERTED := 37,
  /// Analog Output Exceeding Defined Threshold
  ANALOG_OUTPUT_EXCEEDING_DEFINED_THRESHOLD := 40,
  /// Analog Output Falling Below Defined Threshold
  ANALOG_OUTPUT_FALLING_BELOW_DEFINED_THRESHOLD := 41,
  /// Analog Output Exceeding or Falling Below Defined Threshold
  ANALOG_OUTPUT_EXCEEDING_OR_FALLING_BELOW_DEFINED_THRESHOLD := 42,
  /// Analog Output Exceeding or Falling Below Defined Threshold (Inverted)
  ANALOG_OUTPUT_EXCEEDING_OR_FALLING_BELOW_DEFINED_THRESHOLD_INVERTED := 43,
  /// Analog Output Entering Defined Range
  ANALOG_OUTPUT_ENTERING_DEFINED_RANGE := 44,
  /// Analog Output Leaving Defined Range
  ANALOG_OUTPUT_LEAVING_DEFINED_RANGE := 45,
  /// Analog Output Entering or Leaving Defined Range
  ANALOG_OUTPUT_ENTERING_OR_LEAVING_DEFINED_RANGE := 46,
  /// Analog Output Entering or Leaving Defined Range (Inverted)
  ANALOG_OUTPUT_ENTERING_OR_LEAVING_DEFINED_RANGE_INVERTED := 47,
  /// Integer Register Exceeding Defined Threshold
  INTEGER_REGISTER_EXCEEDING_DEFINED_THRESHOLD := 50,
  /// Integer Register Falling Below Defined Threshold
  INTEGER_REGISTER_FALLING_BELOW_DEFINED_THRESHOLD := 51,
  /// Integer Register Exceeding or Falling Below Defined Threshold
  INTEGER_REGISTER_EXCEEDING_OR_FALLING_BELOW_DEFINED_THRESHOLD := 52,
  /// Integer Register Exceeding or Falling Below Defined Value (Inverted)
  INTEGER_REGISTER_EXCEEDING_OR_FALLING_BELOW_DEFINED_VALUE_INVERTED := 53,
  /// Integer Register Entering Defined Range
  INTEGER_REGISTER_ENTERING_DEFINED_RANGE := 54,
  /// Integer Register Leaving Defined Range
  INTEGER_REGISTER_LEAVING_DEFINED_RANGE := 55,
  /// Integer Register Entering or Leaving Defined Range
  INTEGER_REGISTER_ENTERING_OR_LEAVING_DEFINED_RANGE := 56,
  /// Integer Register Entering or Leaving Defined Range (Inverted)
  INTEGER_REGISTER_ENTERING_OR_LEAVING_DEFINED_RANGE_INVERTED := 57,
  /// Real Register Exceeding Defined Threshold
  REAL_REGISTER_EXCEEDING_DEFINED_THRESHOLD := 60,
  /// Real Register Falling Below Defined Threshold
  REAL_REGISTER_FALLING_BELOW_DEFINED_THRESHOLD := 61,
  /// Real Register Exceeding or Falling Below Defined Threshold
  REAL_REGISTER_EXCEEDING_OR_FALLING_BELOW_DEFINED_THRESHOLD := 62,
  /// Real Register Exceeding or Falling Below Defined Threshold (Inverted)
  REAL_REGISTER_EXCEEDING_OR_FALLING_BELOW_DEFINED_THRESHOLD_INVERTED := 63,
  /// Real Register Entering Defined Range
  REAL_REGISTER_ENTERING_DEFINED_RANGE := 64,
  /// Real Register Leaving Defined Range
  REAL_REGISTER_LEAVING_DEFINED_RANGE := 65,
  /// Real Register Entering or Leaving Defined Range
  REAL_REGISTER_ENTERING_OR_LEAVING_DEFINED_RANGE := 66,
  /// Real Register Entering or Leaving Defined Range (Inverted)
  REAL_REGISTER_ENTERING_OR_LEAVING_DEFINED_RANGE_INVERTED := 67
)SINT;
END_TYPE

